FUNCTION_BLOCK Test_HMI (* Service Interface Function Block Type *)
  (* Standard: 61499-2 *)
  (* Version 0.0, 7/14/2016, Andrei, nxtControl GmbH, template *)
  PACKAGE Main;
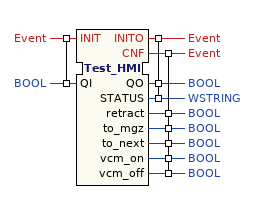
  EVENT_INPUT
    INIT WITH QI;
  END_EVENT
  EVENT_OUTPUT
    INITO WITH QO, STATUS;
    CNF WITH retract, to_mgz, to_next, vcm_on, vcm_off;
  END_EVENT
  VAR_INPUT
    QI : BOOL;
  END_VAR
  VAR_OUTPUT
    QO : BOOL; (* Event Output Qualifier *)
    STATUS : WSTRING; (* Service Status *)
    retract : BOOL;
    to_mgz : BOOL;
    to_next : BOOL;
    vcm_on : BOOL;
    vcm_off : BOOL;
  END_VAR
END_FUNCTION_BLOCK
